(* CoDeSys 2.3 export: GETIPADDRESS.EXP *)

(* POU Udp specific/GetIPAddress, ST *)
FUNCTION GetIPAddress : DINT
VAR_INPUT
	stIPAddress:STRING;		(* IP-address or computer name *)
END_VAR
VAR
	diIPAddress:DINT;
END_VAR
(* @TEXT_IMPLEMENTATION := 'ST' *)
diIPAddress := SysSockInetAddr(stIPAddress);
IF (stIPAddress = '255.255.255.255') THEN
	(*Avoid name-resolution on our default broadcast address.*)
	GetIPAddress:=diIPAddress;
	RETURN ;
END_IF
IF diIPAddress = SOCKET_INADDR_NONE THEN
	diIPAddress := SysSockGetHostByName(ADR(stIPAddress));
END_IF
GetIPAddress:=diIPAddress;
END_FUNCTION
